INTERFACE IComponent

PROPERTY Lock : INT
GET
END_GET
SET
END_SET
END_PROPERTY

END_INTERFACE

(* stored: Version 1.1.0.1, ProductVersion 3.1.4024.5
   Itf IComponent: Id {1d4a5c73-6248-441d-aaab-9bd8b4ee3caf}
   Property Lock: Id {e00a820b-feed-4fbe-9eb9-03dbb5f0f825}
   Get Get: Id {95b9a86e-3519-468c-91ee-bd964e77bfe1}
   Set Set: Id {9097b4fa-f009-4534-a3db-e3ad0723b86c} *)
